Fanuc KAREL source: kc00026.KL

-- PROVISIONAL review KL for V770-1; original PC SHA256 92714327e0748cbf6dd9bf451a4a4a5cfb11713ea6b81bc284c193a4890ecd52
-- Incomplete behavior may be omitted. Consult companion uncertainty JSON. Do not deploy.
PROGRAM KC00026
%NOLOCKGROUP
BEGIN
  -- UNRESOLVED_PC offsets 5-45; opcodes 27,22,22,22,22,22,22,31
  -- UNRESOLVED_PC offsets 50-54; opcodes 7F
END KC00026
